TYPE E_VCN :
	(
CloseValve	:= 0,
ControlValve	:= 1,
OpenValve	:= 2
	);
END_TYPE

(* stored: Version 1.1.0.1, ProductVersion 3.1.4018.5
   DUT E_VCN: Id {8cba8144-9517-4b79-93a4-dc42ff0eaf7b} *)
